Fanuc KAREL source: compact_preamble.KL

PROGRAM KB00141
%NOLOCKGROUP
%ENVIRONMENT FDEV
VAR
P1 : STRING[80];P2:INTEGER
BEGIN
P1='A'
P2=1
PURGE_DEV(P1,P2)
END KB00141
